FUNCTION_BLOCK EventRunner
VAR_INPUT
  save_data_to_file: BOOL;
END_VAR
VAR_OUTPUT
END_VAR
VAR
  event_id_counter: INT;
  localtime: FB_LocalSystemTime := (bEnable:=TRUE);
  actSystemTime: TIMESTRUCT;
  event_history_counter: INT;
  disable_ads_output: BOOL;
  event_logger: ARRAY [1..Properties.NUM_LOGGER] OF EventLogger;
  act_logger_counter: INT;
END_VAR

(* 
der runner wird am ende des sps programms ausgefuehrt
- als input kommt das signal zum sichern der daten (bei der cx81xx bspw. das signal der usv). diese werden binaer gesichtert, koennen jedoch zusaetzlich als csv gesichert werden
- ansonsten kuemmert sich der runner nur um die erstellung eines arrays zur darstellung in einer hmi mit den aktuell aktiven events
- im programm werden pro meldung event-instanzen erstellt. diese regestrieren sich selbst. die richtige id wird der pfad zur instanzvariable sein
- im runner wird zudem das datum immer aktualisiert
*)

PROPERTY act_time : TIMESTRUCT
GET
IF time_valid THEN
  act_time := localtime.systemTime;
END_IF
END_GET
END_PROPERTY

METHOD add_logger
VAR_INPUT
  logger: EventLogger;
END_VAR
IF act_logger_counter < Properties.NUM_LOGGER AND ADR(logger) <> 0 THEN
  act_logger_counter := act_logger_counter + 1;
  event_logger[act_logger_counter] := logger;
END_IF
END_METHOD

METHOD add_message
VAR_INPUT
  id: INT;
  message: STRING(255);
  level: EventLevel;
END_VAR
inc_history_counter();

GVL_EventLogger.event_history[event_history_counter].id := id;
GVL_EventLogger.event_history[event_history_counter].level := level;
GVL_EventLogger.event_history[event_history_counter].timestamp_raised := act_time;
GVL_EventLogger.event_history[event_history_counter].timestamp_cleared := act_time;

ads_log(id:=id, message:=message, level:=level);
END_METHOD

METHOD ads_log
VAR_INPUT
  id: INT;
  message: STRING(255);
  level: EventLevel;
END_VAR
VAR
  mask: DWORD;
  prefix: STRING(12);
  formatted_message: STRING(255);
  event_pointer: POINTER TO FBEvent;
END_VAR
IF disable_ads_output THEN
  RETURN;
END_IF

CASE level OF
EventLevel.INFO:
  mask := ADSLOG_MSGTYPE_HINT OR ADSLOG_MSGTYPE_LOG;
  prefix := ' | Info: ';
EventLevel.WARNING:
  mask := ADSLOG_MSGTYPE_WARN OR ADSLOG_MSGTYPE_LOG;
  prefix := ' | Warnung: ';
EventLevel.ERROR:
  mask := ADSLOG_MSGTYPE_ERROR OR ADSLOG_MSGTYPE_LOG;
  prefix := ' | Fehler: ';
ELSE
  mask := ADSLOG_MSGTYPE_HINT OR ADSLOG_MSGTYPE_LOG;
  prefix := ' | Info: ';
END_CASE

formatted_message := CONCAT(prefix, message);
//message := CONCAT(event_pointer^.instance_path, message);

ADSLOGSTR(mask, formatted_message, '');
END_METHOD

METHOD clear_alarm
VAR_INPUT
  id: INT;
END_VAR
VAR
  count: INT;
END_VAR
count := raised_history_count(id:=id);
IF count > 0 THEN
  GVL_EventLogger.event_history[count].timestamp_cleared := act_time;
END_IF
END_METHOD

METHOD INTERNAL generate_event_id : INT
VAR_INPUT
END_VAR
event_id_counter := event_id_counter + 1;
// TODO: add conditional for max num
generate_event_id := event_id_counter;
END_METHOD

METHOD inc_history_counter
VAR_INPUT
END_VAR
event_history_counter := LIMIT(1, event_history_counter + 1, Properties.NUM_EVENT_HISTORY);
END_METHOD

METHOD raise_alarm
VAR_INPUT
  id: INT;
  message: STRING(255);
  level: EventLevel;
END_VAR
VAR
  undefined_time: TIMESTRUCT;
END_VAR
IF raised_history_count(id:=id) = 0 THEN
  inc_history_counter();
  GVL_EventLogger.event_history[event_history_counter].id := id;
  GVL_EventLogger.event_history[event_history_counter].level := level;
  GVL_EventLogger.event_history[event_history_counter].timestamp_raised := act_time;
  GVL_EventLogger.event_history[event_history_counter].timestamp_cleared := undefined_time;
  
  ads_log(id:=id, message:=message, level:=level);
END_IF
END_METHOD

METHOD raised_history_count : INT
VAR_INPUT
  id: INT;
END_VAR
VAR
  i: INT;
  undefined_time: TIMESTRUCT;
END_VAR
FOR i:=1 TO Properties.NUM_EVENT_HISTORY DO
  IF GVL_EventLogger.event_history[i].id = id AND timestruct_equal(GVL_EventLogger.event_history[i].timestamp_cleared, undefined_time) THEN
    raised_history_count := i;
    EXIT;
	END_IF
END_FOR
END_METHOD

METHOD run
VAR_INPUT
  disable_ads_output: BOOL; // for testing purposes
END_VAR
VAR
  read_done: BOOL;
  error_id: UDINT;
END_VAR
localtime();
THIS^.disable_ads_output := disable_ads_output;

save_logger(execute:=save_data_to_file);
END_METHOD

METHOD save_logger
VAR_INPUT
  execute: BOOL;
END_VAR
VAR
  i: INT;
END_VAR
FOR i:=1 TO act_logger_counter DO
  IF ADR(event_logger[i]) <> 0 THEN
    event_logger[i].save(
      execute:=execute,
      data_ptr:=ADR(GVL_EventLogger.event_history),
      data_size:=SIZEOF(GVL_EventLogger.event_history));
  END_IF
END_FOR
END_METHOD

PROPERTY time_valid : BOOL
GET
time_valid := localtime.bValid;
END_GET
END_PROPERTY

METHOD timestruct_equal : BOOL
VAR_INPUT
  timestruct_1: TIMESTRUCT;
  timestruct_2: TIMESTRUCT;
END_VAR
timestruct_equal := timestruct_1.wDay = timestruct_2.wDay;
timestruct_equal := timestruct_equal AND timestruct_1.wDayOfWeek = timestruct_2.wDayOfWeek;
timestruct_equal := timestruct_equal AND timestruct_1.wHour = timestruct_2.wHour;
timestruct_equal := timestruct_equal AND timestruct_1.wMilliseconds = timestruct_2.wMilliseconds;
timestruct_equal := timestruct_equal AND timestruct_1.wMinute = timestruct_2.wMinute;
END_METHOD

END_FUNCTION_BLOCK

(* stored: Version 1.1.0.1, ProductVersion 3.1.4022.18
   POU EventRunner: Id {0d525c38-ad3f-47ea-a798-0db63d693ea9}, SpecialFunc None
   Property act_time: Id {7e8ceabb-80c4-4035-9e65-42491c23b792}
   Get Get: Id {380360c5-f864-458f-9b41-ca220d584c69}
   Method add_logger: Id {2651f9dc-bec6-4584-8fd4-83f95233f0d4}
   Method add_message: Id {f126ae69-dbb0-4036-b829-819771f00c85}
   Method ads_log: Id {0c503934-a332-47a9-ab84-e19746f835d8}
   Method clear_alarm: Id {07a3255c-8c06-4ac3-9bc3-7cc05616380c}
   Method generate_event_id: Id {45e6113d-bd59-45d0-baac-1654e214698c}
   Method inc_history_counter: Id {c1bf2e16-ba4b-408b-a3aa-157cc3fb0417}
   Method raise_alarm: Id {b9a7897e-9e09-4385-9cb5-c61ebd939157}
   Method raised_history_count: Id {2dd42452-2a07-452a-9647-430f1f9f8d83}
   Method run: Id {8739a071-bf84-4818-9cb8-125145dee33b}
   Method save_logger: Id {da433036-a647-4f83-9bab-6401224e9fee}
   Property time_valid: Id {97759346-09f2-489b-abe8-e35197fe4275}
   Get Get: Id {0bd76518-28fe-433e-82d9-2b30ff8be461}
   Method timestruct_equal: Id {d3110f90-c794-4c07-a338-1efa49783308} *)
